{attribute 'GeneratedUsingTerminal: EL6900-0000-0016'}
{attribute addProperty BoxType "EL6900-0000-0016"}
{attribute addProperty Id "Safety_Project_StateAT %I*BYTE1Login_ActiveAT %I*BOOL1Input_Size_MismatchAT %I*BOOL1Output_Size_MismatchAT %I*BOOL1TxPDO_StateAT %I*BOOL1TxPDO_ToggleAT %I*BOOL1"}
{attribute addProperty CRC "1952193002"}
{attribute addProperty Size "6"}
TYPE DEVICE_Inputs_745C19EA :
STRUCT
	{attribute addProperty Name "Safety_Project_State"}
	Safety_Project_State AT %I* : BYTE;
	{attribute addProperty Name "Login_Active"}
	Login_Active AT %I* : BOOL;
	{attribute addProperty Name "Input_Size_Mismatch"}
	Input_Size_Mismatch AT %I* : BOOL;
	{attribute addProperty Name "Output_Size_Mismatch"}
	Output_Size_Mismatch AT %I* : BOOL;
	{attribute addProperty Name "TxPDO_State"}
	TxPDO_State AT %I* : BOOL;
	{attribute addProperty Name "TxPDO_Toggle"}
	TxPDO_Toggle AT %I* : BOOL;
END_STRUCT
END_TYPE

(* stored: Version 1.2.0.0, ProductVersion 3.1.4024.9
   DUT DEVICE_Inputs_745C19EA: Id {55d79724-471f-415d-828c-cbb9aa1d9f46} *)
